# B&R Automation Studio project LampTest
Automation Studio 6.0.1.886; technology packages: OpcUaCs 6.0.0

## Configuration Config1

CPU X20CP1686X, AutomationRuntime 6.0.7000, Build 11.3.0, Vc 6.0.7000

### Task classes (Cpu.sw)
```
Cyclic#4:
  lampTest <- lampTest.prg
```

### Hardware
```
X20CP1686X : X20CP1686X v1.8.0.0
  Connector IF2:
    ActivateDevice = 1
  ConfigurationID = LampTest_Config1
  Simulation = 1
  FileDevice1
  FileDeviceName1 = USER
  FileDevicePath1 = USER_PATH
```

## Logical view

### Program Logical/lampTest (IEC)

#### Cyclic.ld - Cyclic code
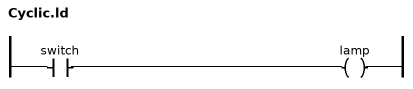
Diagram, in the editor's own instruction-list form stored in the file:
```il
PROGRAM _CYCLIC

{NetworkNumber := 1}
LD	switch
ST	lamp

END_PROGRAM
```

#### Init.ld - Initialization code
Diagram, in the editor's own instruction-list form stored in the file:
```il
PROGRAM _INIT

END_PROGRAM
```

#### Exit.ld - Exit code
Diagram, in the editor's own instruction-list form stored in the file:
```il
PROGRAM _EXIT

END_PROGRAM
```

#### Variables.var - Local variables
```iecst
VAR
	switch : BOOL;
	lamp : BOOL;
END_VAR
```

Listed in the project but not available here: Logical/Global.typ, Logical/Libraries, Logical/lampTest/Types.typ
